// TIA Portal V15.1 export
// export: Created 2020-06-12T07:35:44.8193359Z, ExportSetting None, DisplayName Totally Integrated Automation Portal, DisplayVersion V15.1, DisplayName TIA Portal Openness, DisplayVersion V15.1, DisplayName STEP 7 Professional, DisplayVersion V15.1, DisplayName STEP 7 Safety, DisplayVersion V15.1, DisplayName WinCC Advanced, DisplayVersion V15.1
FUNCTION "MS1_CLAMP" : Void   // FC951, FBD
TITLE = Program for open/close Baseplate Clamp Meltstation 1
{ S7_Optimized_Access := 'FALSE' }
// stored: AutoNumber false, SetENOAutomatically False
   VAR_TEMP
      _ls_opn : Bool;
      tClose1 : Bool;
      tOpen1 : Bool;
      _csf : Bool;
      _ps01_ton : Bool;
      tExtClose : Bool;
      tExtOpen : Bool;
      tClose2 : Bool;
      tOpen2 : Bool;
   END_VAR
BEGIN

REGION Network 1: common system fault
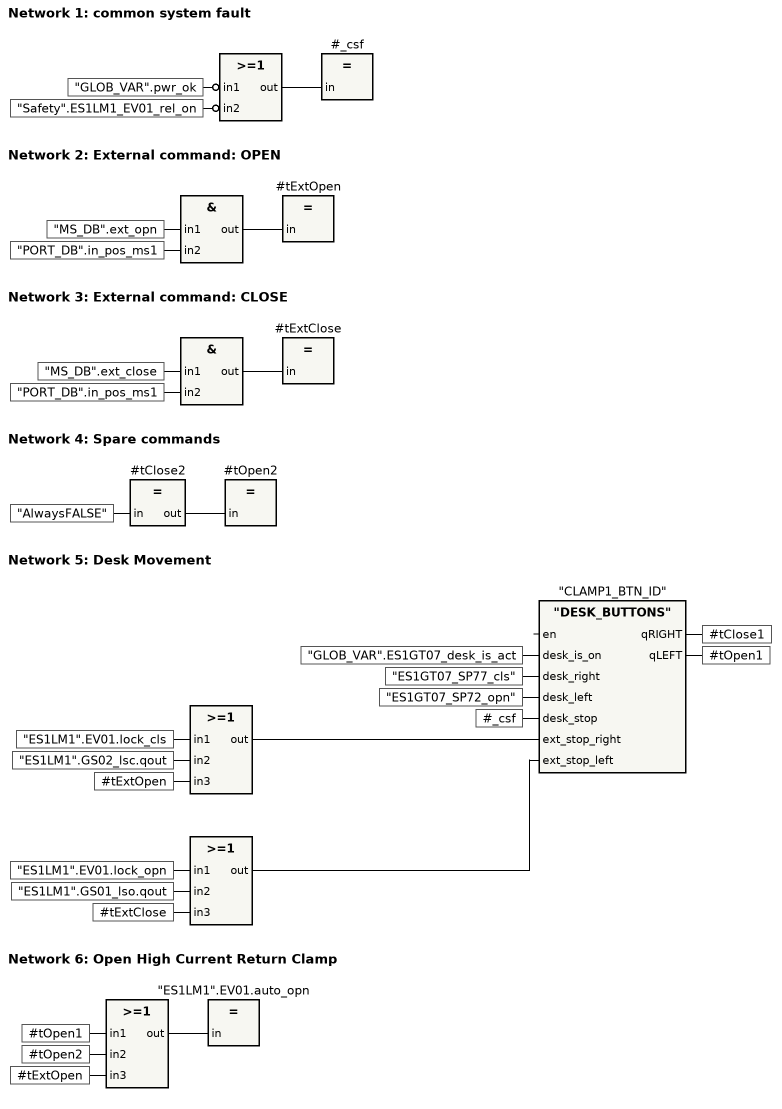
   #_csf := NOT "GLOB_VAR".pwr_ok OR NOT "Safety".ES1LM1_EV01_rel_on;
END_REGION

REGION Network 2: External command: OPEN
   #tExtOpen := "MS_DB".ext_opn AND "PORT_DB".in_pos_ms1;
END_REGION

REGION Network 3: External command: CLOSE
   #tExtClose := "MS_DB".ext_close AND "PORT_DB".in_pos_ms1;
END_REGION

REGION Network 4: Spare commands
   #tClose2 := "AlwaysFALSE";
   #tOpen2 := "AlwaysFALSE";
END_REGION

REGION Network 5: Desk Movement
   "CLAMP1_BTN_ID"(desk_is_on := "GLOB_VAR".ES1GT07_desk_is_act,   // "DESK_BUTTONS"
                   desk_right := "ES1GT07_SP77_cls",
                   desk_left := "ES1GT07_SP72_opn",
                   desk_stop := #_csf,
                   ext_stop_right := "ES1LM1".EV01.lock_cls OR "ES1LM1".GS02_lsc.qout OR #tExtOpen,
                   ext_stop_left := "ES1LM1".EV01.lock_opn OR "ES1LM1".GS01_lso.qout OR #tExtClose,
                   qRIGHT => #tClose1,
                   qLEFT => #tOpen1);
END_REGION

REGION Network 6: Open High Current Return Clamp
   "ES1LM1".EV01.auto_opn := #tOpen1 OR #tOpen2 OR #tExtOpen;
END_REGION

REGION Network 7: Close High Current Return Clamp
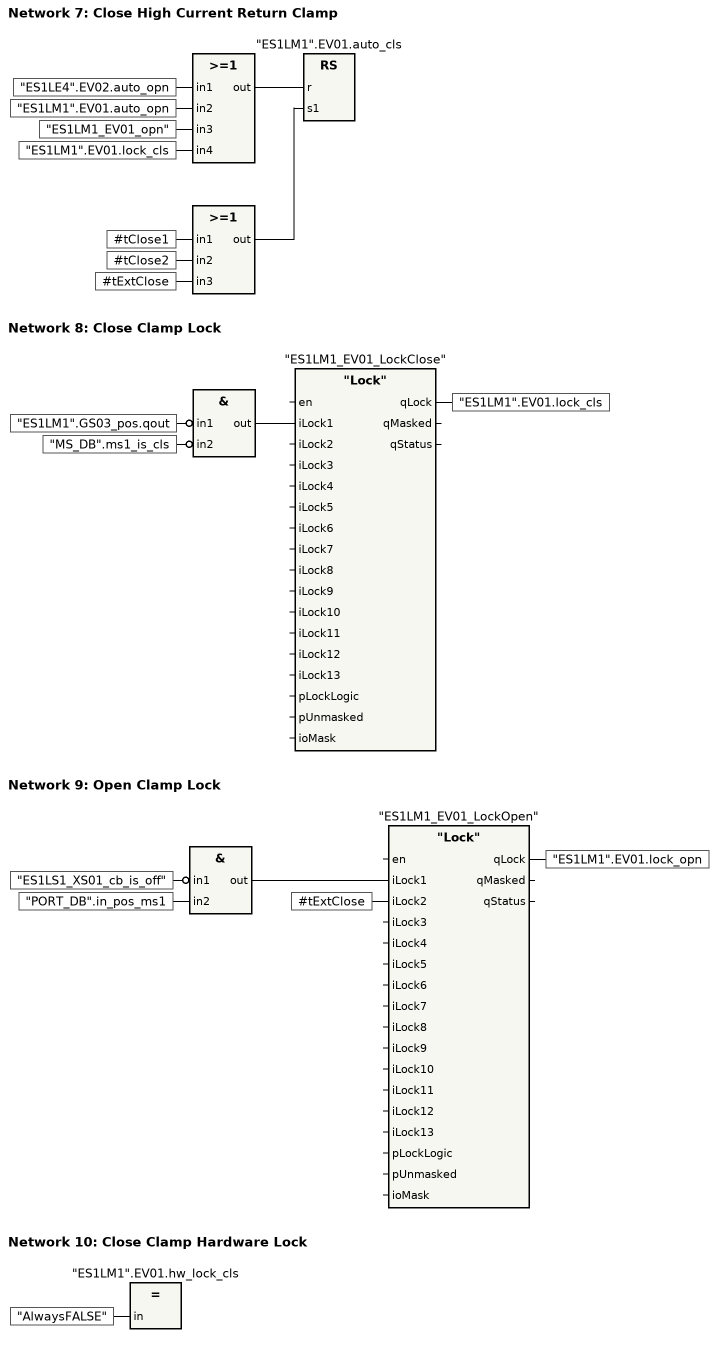
   IF "ES1LE4".EV02.auto_opn OR "ES1LM1".EV01.auto_opn OR "ES1LM1_EV01_opn" OR "ES1LM1".EV01.lock_cls THEN
       "ES1LM1".EV01.auto_cls := FALSE;   // RS flip-flop
   END_IF;
   IF #tClose1 OR #tClose2 OR #tExtClose THEN "ES1LM1".EV01.auto_cls := TRUE; END_IF;
END_REGION

REGION Network 8: Close Clamp Lock
   "ES1LM1_EV01_LockClose"(iLock1 := NOT "ES1LM1".GS03_pos.qout AND NOT "MS_DB".ms1_is_cls,   // "Lock"
                           qLock => "ES1LM1".EV01.lock_cls);
END_REGION

REGION Network 9: Open Clamp Lock
   "ES1LM1_EV01_LockOpen"(iLock1 := NOT "ES1LS1_XS01_cb_is_off" AND "PORT_DB".in_pos_ms1,   // "Lock"
                          iLock2 := #tExtClose,
                          qLock => "ES1LM1".EV01.lock_opn);
END_REGION

REGION Network 10: Close Clamp Hardware Lock
   "ES1LM1".EV01.hw_lock_cls := "AlwaysFALSE";
END_REGION

REGION Network 11: Open Clamp Hardware Lock
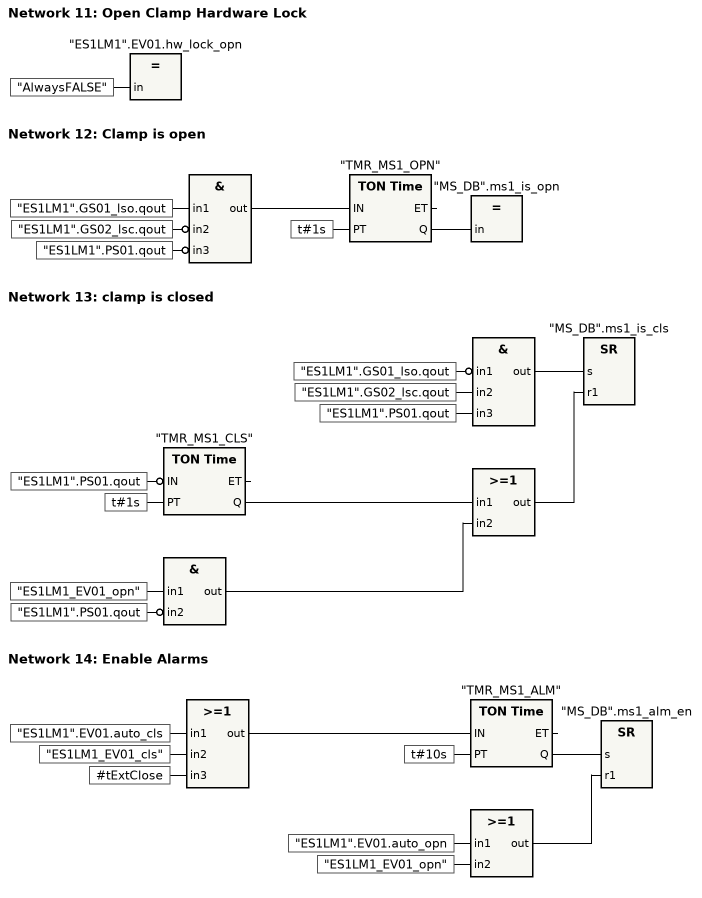
   "ES1LM1".EV01.hw_lock_opn := "AlwaysFALSE";
END_REGION

REGION Network 12: Clamp is open
   "TMR_MS1_OPN".TON(IN := "ES1LM1".GS01_lso.qout AND NOT "ES1LM1".GS02_lsc.qout AND NOT "ES1LM1".PS01.qout,
                     PT := t#1s);
   "MS_DB".ms1_is_opn := "TMR_MS1_OPN".Q;
END_REGION

REGION Network 13: clamp is closed
   "TMR_MS1_CLS".TON(IN := NOT "ES1LM1".PS01.qout, PT := t#1s);
   IF NOT "ES1LM1".GS01_lso.qout AND "ES1LM1".GS02_lsc.qout AND "ES1LM1".PS01.qout THEN
       "MS_DB".ms1_is_cls := TRUE;   // SR flip-flop
   END_IF;
   IF "TMR_MS1_CLS".Q OR ("ES1LM1_EV01_opn" AND NOT "ES1LM1".PS01.qout) THEN
       "MS_DB".ms1_is_cls := FALSE;
   END_IF;
END_REGION

REGION Network 14: Enable Alarms
   "TMR_MS1_ALM".TON(IN := "ES1LM1".EV01.auto_cls OR "ES1LM1_EV01_cls" OR #tExtClose, PT := t#10s);
   IF "TMR_MS1_ALM".Q THEN
       "MS_DB".ms1_alm_en := TRUE;   // SR flip-flop
   END_IF;
   IF "ES1LM1".EV01.auto_opn OR "ES1LM1_EV01_opn" THEN "MS_DB".ms1_alm_en := FALSE; END_IF;
END_REGION
END_FUNCTION
